(* CODESYS project WashingMachine.project

Project tree, tasks and I/O mapping:
  Device : CODESYS Control Win V3, CODESYS, version 3.5.20.0
    application Application
      libraries: Standard, 3.5.18.0 (System); VisuDialogs, * (System)
      task MainTask (cyclic, interval t#20ms, priority 1) calls Simulation_Program
      task VISU_TASK (cyclic, interval 100 ms, priority 31) calls VisuElems.Visu_Prg
      visualisation Visualization
      global variables GVL
      program Simulation_Program [ST]
  text list GlobalTextList
*)

// Device/Application/GVL
{attribute 'qualified_only'}
VAR_GLOBAL
	temperature		: INT;		 	(*Sensor: current temperature of the water*)
	soaplevel		: INT; 			(*Sensor: current soap level*)
	waterlevel		: INT;			(*Sensor: current water level*)
	prog_number		: INT;			(*Input: program selected by the user*)
	temp_number		: INT; 			(*Input: temperature selected by the user*)
	run				: BOOL;			(*Input: if TRUE the washing machine works*)
	fillsoap		: BOOL; 		(*Input: if TRUE the soap tray is full*)
	bulls_eye_open	: BOOL := TRUE;	(*Input: if TRUE the door is open*)

	hot				: BOOL;			(*Actuator: if TRUE the resistor turns on*)
	motor_on		: BOOL;			(*Actuator: if TRUE the basket motor is turned on*)
	bulls_eye_lock	: BOOL;			(*Actuator: if TRUE the Door is locked*)
	emptysoap		: BOOL;			(*Actuator: if TRUE the soap tray is emptied*)
	fillwater		: BOOL;			(*Actuator: if TRUE the water is added*)
	emptywater		: BOOL;			(*Actuator: if TRUE the water is drained*)

	heat_alarm		: BOOL; 		(*Visualization: if TRUE alerts the user of the resistor fault*)
	water_in_alarm	: BOOL;			(*Visualization: if TRUE alerts the user of the water intake valve fault*)
	water_out_alarm	: BOOL; 		(*Visualization: if TRUE alerts the user of the water drain valve fault*)
	soap_alarm		: BOOL;			(*Visualization: if TRUE there is no soap*)
	prog_error		: BOOL;			(*Visualization: if TRUE the program selected is wrong*)
	temp_error		: BOOL;			(*Visualization: if TRUE the temperature selected is wrong*)
	rinse			: BOOL; 		(*Visualization: if TRUE the rinsing operation is going on*)
	prewash			: BOOL; 		(*Visualization: if TRUE the prewashing operation is going on*)
	wash			: BOOL; 		(*Visualization: if TRUE the washing operation is going on*)

	motor			: INT;			(*Only for simulation: angular position of the basket*)
	heat_fail		: BOOL;			(*Only for simulation: if TRUE the resistor cannot turn on*)
	water_in_fail	: BOOL;			(*Only for simulation: if TRUE the water intake valve is faulty*)
	water_out_fail	: BOOL;			(*Only for simulation: if TRUE the water drain valve is faulty*)
END_VAR

// Device/Application/Simulation_Program
PROGRAM Simulation_Program
VAR
		bulls_eye_open_past	:BOOL := TRUE;
END_VAR

(*Temperature value simulation*)
IF ((GVL.hot)AND(NOT GVL.heat_fail)) THEN 
	GVL.temperature := GVL.temperature + 1;
ELSE
	GVL.temperature := GVL.temperature - 1;
END_IF

IF GVL.temperature > 100 THEN 
	GVL.temperature := 100;
END_IF

IF GVL.temperature < 0 THEN 
	GVL.temperature := 0;
END_IF


(*Soap level simulation*)
IF GVL.fillsoap THEN 
	GVL.soaplevel := GVL.soaplevel + 5;
ELSIF GVL.emptysoap THEN 
	GVL.soaplevel := GVL.soaplevel - 3;
END_IF

IF GVL.soaplevel >= 50 THEN 
	GVL.soaplevel := 50;
	GVL.fillsoap := FALSE;
END_IF

IF GVL.soaplevel < 0 THEN 
	GVL.soaplevel := 0;
END_IF


(*Door state simulation*)
IF ((GVL.bulls_eye_open <> bulls_eye_open_past)AND(NOT GVL.bulls_eye_lock)) THEN 
	bulls_eye_open_past := GVL.bulls_eye_open ;
ELSIF GVL.bulls_eye_lock THEN
	GVL.bulls_eye_open := bulls_eye_open_past;
END_IF


(*Water level simulation*)
IF ((GVL.fillwater)AND(NOT GVL.water_in_fail)) THEN 
	GVL.waterlevel := GVL.waterlevel + 2;
ELSIF ((GVL.emptywater)AND(NOT GVL.water_out_fail)) THEN
	GVL.waterlevel := GVL.waterlevel - 4;
END_IF

IF GVL.waterlevel > 150 THEN 
	GVL.waterlevel := 150;
END_IF

IF GVL.waterlevel < 0 THEN 
	GVL.waterlevel := 0;
END_IF


(*Motor simulation*)
IF (GVL.motor_on) THEN 
	GVL.motor := GVL.motor + 10;
END_IF

IF GVL.motor > 360 THEN 
	GVL.motor := 0;
END_IF

END_PROGRAM

// Device/Application/Visualization
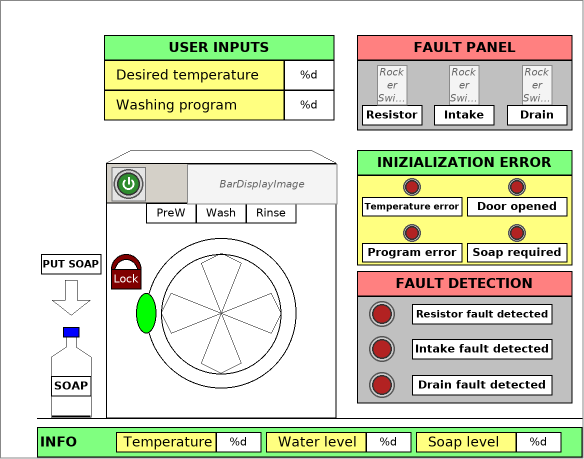
VISUALIZATION Visualization  // 584x459
    Line (37,418) (582,418)
    Rectangle (106,178 230x240)
    Ellipse (162,254 118x118)
    Rectangle (161,255 120x120)
        p1126004900: -GVL.waterlevel/3*2
    Ellipse (146,238 150x150)
    Ellipse (161,254 120x120)
    Polygon (221,253) (201,263) (221,313) (171,293) (161,313) (171,333) (221,313) (201,363) (221,373) (241,363) (221,313) (271,333) (281,313) (271,293) (221,313) (241,263)
        p2858320360: GVL.motor
    Ellipse (136,293 20x40), colour toggle: GVL.bulls_eye_open
        toggle GVL.bulls_eye_open
    Ellipse (111,254 30x30), colour toggle: GVL.bulls_eye_lock
    Ellipse (114,259 24x27)
    Rectangle (111,269 30x20), "Lock", colour toggle: GVL.bulls_eye_lock
    Rectangle (106,163 230x40)
    Rectangle (146,203 50x20), "PreW", colour toggle: GVL.prewash
    Rectangle (196,203 50x20), "Wash", colour toggle: GVL.wash
    Rectangle (246,203 50x20), "Rinse", colour toggle: GVL.rinse
    Polygon (106,163) (131,150) (311,150) (336,163)
    PowerSwitch (111,167 35x34), variable: GVL.run, behaviour: TOGGLE, style: Switch-PowerSwitch-Green
    BarDisplayImage (187,164 150x40), value: GVL.temperature, style: BarDisplayImage-Gray, scale format: %.0f, scale 0..90
    Polygon (51,417) (51,357) (66,347) (66,332) (76,332) (76,347) (91,357) (91,417)
    Rectangle (63,327 16x10)
    Rectangle (104,60 180x30), "Desired temperature"
        OnMouseDown: write GVL.temp_number via VisuDialogs.Numpad, min 0, max 100, format 0
    Rectangle (104,90 180x30), "Washing program"
        OnMouseDown: write GVL.prog_number via VisuDialogs.Numpad, min 0, max 100, format 0
    Rectangle (104,35 230x25), "USER INPUTS"
    Rectangle (284,60 50x30), "%d", text variable: GVL.temp_number
    Rectangle (284,90 50x30), "%d", text variable: GVL.prog_number
    Rectangle (37,427 545x30), "INFO"
    Rectangle (116,432 100x20), "Temperature"
    Rectangle (357,150 215x25), "INIZIALIZATION ERROR"
    Rectangle (216,432 45x20), "%d", text variable: GVL.temperature
    Rectangle (266,432 100x20), "Water level"
    Rectangle (366,432 45x20), "%d", text variable: GVL.waterlevel
    Rectangle (416,432 100x20), "Soap level"
    Rectangle (516,432 45x20), "%d", text variable: GVL.soaplevel
    Rectangle (357,175 215x90)
    Lamp1 (402,177 20x20), variable: GVL.temp_error, style: Lamp-Lamp1-Red
    Rectangle (362,197 100x19), "Temperature error"
    Lamp1 (507,177 20x20), variable: GVL.bulls_eye_open, style: Lamp-Lamp1-Red
    Rectangle (467,197 100x19), "Door opened"
    Lamp1 (402,223 20x20), variable: GVL.prog_error, style: Lamp-Lamp1-Red
    Rectangle (362,243 100x19), "Program error"
    Lamp1 (507,223 20x20), variable: GVL.soap_alarm, style: Lamp-Lamp1-Red
    Rectangle (467,243 100x19), "Soap required"
    Rectangle (357,35 215x25), "FAULT PANEL"
    Rectangle (357,60 215x70)
    Rectangle (362,105 60x20), "Resistor"
    RockerSwitch (377,65 30x40), variable: GVL.heat_fail, behaviour: TOGGLE, style: Switch-RockerSwitch-Red
    RockerSwitch (449,65 30x40), variable: GVL.water_in_fail, behaviour: TOGGLE, style: Switch-RockerSwitch-Red
    Rectangle (434,105 60x20), "Intake"
    RockerSwitch (522,65 30x40), variable: GVL.water_out_fail, behaviour: TOGGLE, style: Switch-RockerSwitch-Red
    Rectangle (507,105 60x20), "Drain"
    Rectangle (357,271 215x25), "FAULT DETECTION"
    Rectangle (357,296 215x107)
    Lamp1 (367,299 30x30), variable: GVL.heat_alarm, style: Lamp-Lamp1-Red
    Rectangle (412,304 140x20), "Resistor fault detected"
    Lamp1 (367,370 30x30), variable: GVL.water_out_alarm, style: Lamp-Lamp1-Red
    Lamp1 (367,334 30x30), variable: GVL.water_in_alarm, style: Lamp-Lamp1-Red
    Rectangle (412,339 140x20), "Intake fault detected"
    Rectangle (412,375 140x20), "Drain fault detected"
    Rectangle (52,416 38x0)
        p2773130477: -GVL.soaplevel
    Rectangle (51,376 40x20), "SOAP"
    Polygon (65,280) (65,300) (52,300) (71,315) (90,300) (77,300) (77,280), colour toggle: GVL.fillsoap
        toggle GVL.fillsoap
    Rectangle (41,254 60x20), "PUT SOAP"
END_VISUALIZATION
